Fanuc KAREL source: ka00010.KL

PROGRAM KA00010
%STACKSIZE=65535
%PRIORITY=65535
%NOLOCKGROUP
VAR
SRC : INTEGER
-- UNRESOLVED DECLARATIONS (source type spelling not recovered)
-- DST : TYPE_0x001C (type_u16=0x001C)
BEGIN
SRC=2
DST=SRC
END KA00010
